{attribute 'enable_dynamic_creation'}
{attribute 'no_explicit_call' := 'Singleton is a CLASS and must be accessed using methods or properties'}
FUNCTION_BLOCK MessageLoggerSingleton IMPLEMENTS I_MessageLogger // USE MessageLogger!!
VAR
	_message			: STRING;
END_VAR

METHOD LogMessage : STRING
VAR_INPUT
	message			: STRING;
END_VAR
_message := message;
END_METHOD

{warning 'add property implementation'}
PROPERTY message : STRING
GET
message  := _message;
END_GET
END_PROPERTY

END_FUNCTION_BLOCK

(* stored: Version 1.1.0.1, ProductVersion 3.1.4024.11
   POU MessageLoggerSingleton: Id {1b3b14f1-e859-411d-8a61-143a2d245380}, SpecialFunc None
   Method LogMessage: Id {f8faff62-0ffe-4874-8d15-d05f819a7ee1}
   Property message: Id {5619e4e7-2180-4d80-8812-68d9458f0fb9}
   Get Get: Id {44bc55b8-7b5b-416c-a6ac-373ae3646477} *)
